(* IEC 61131-3 sources: SJ_AGV/PLC/Standard_functions.4.4.0/DataUpload, 2 files *)

(* ---- DataUpload_FB.ST ---- *)
FUNCTION_BLOCK DataUpload_FB
VAR_EXTERNAL
ndc8 : NDC8_T;

UploadData_ModBus_ValueWord:ARRAY[1..500] OF Word;
UploadData_ModBus_ValueBOOL:ARRAY[1..400] OF BOOL;

ConvWord:WORD;			(*Sum of the two first bytes*)

ConvByteL:Byte;			(*Low byte*)
ConvByteH:Byte;			(*High byte*)

ConvBit0:BOOL;			(*		 1 	    *)
ConvBit1:BOOL;			(*		 2 		*)
ConvBit2:BOOL;			(*		 4 		*)
ConvBit3:BOOL;			(*		 8 		*)
ConvBit4:BOOL;			(*	    10 		*)
ConvBit5:BOOL;			(*	    20 		*)
ConvBit6:BOOL;			(*	    40 		*)
ConvBit7:BOOL;          (*	    80 		*)
ConvBit8:BOOL;			(*		100     *)
ConvBit9:BOOL;			(*		200 	*)
ConvBit10:BOOL;			(*		400  	*)
ConvBit11:BOOL;			(*		800 	*)
ConvBit12:BOOL;			(*	   1000 	*)
ConvBit13:BOOL;			(*	   2000 	*)
ConvBit14:BOOL;			(*	   4000 	*)
ConvBit15:BOOL;         (*	   8000 	*)

(*BeijerSetParameters:BeijerSetParameters_T;*)

END_VAR

VAR_INPUT

END_VAR

VAR_OUTPUT

END_VAR

VAR

Angle_DINT : DINT;
Angle_REAL : REAL;

DataUpload : DataUpload_ModbusTCPIP_FB;

END_VAR
(****************************************************************************)

(* Update Data *)

(* Scanner_x *)
ConvDINT := NDC8.LS2000.X;
UploadData_ModBus_ValueWord [2]:=ConvWord2;
UploadData_ModBus_ValueWord [1]:=ConvWord;

(* Scanner_y *)
ConvDINT := NDC8.LS2000.Y;
UploadData_ModBus_ValueWord [4]:=ConvWord2;
UploadData_ModBus_ValueWord [3]:=ConvWord;

(* Scanner_t *)
Angle_REAL := NDC8.LS2000.Angle * 100.0;
Angle_DINT := REAL_TO_DINT(Angle_REAL);

ConvDINT := Angle_DINT;
UploadData_ModBus_ValueWord [6]:=ConvWord2;
UploadData_ModBus_ValueWord [5]:=ConvWord;

(* Max Speed *)
ConvDINT := NDC8.Vehicle.MaxSpeed;
UploadData_ModBus_ValueWord [8]:=ConvWord2;
UploadData_ModBus_ValueWord [7]:=ConvWord;

(* Enc1Scal *)
ConvUDINT := NDC8.DCD_6.SteerEncScale;
UploadData_ModBus_ValueWord [10]:=ConvWord2;
UploadData_ModBus_ValueWord [9]:=ConvWord;

(* Enc1Offs *)
ConvDINT := INT_TO_DINT(NDC8.DCD_6.SteerEncOffset);
UploadData_ModBus_ValueWord [12]:=ConvWord2;
UploadData_ModBus_ValueWord [11]:=ConvWord;

(* Enc3Scal *)
ConvUDINT := NDC8.DCD_8.SteerEncScale;
UploadData_ModBus_ValueWord [14]:=ConvWord2;
UploadData_ModBus_ValueWord [13]:=ConvWord;

(* Enc3Offs *)
ConvDINT := INT_TO_DINT(NDC8.DCD_8.SteerEncOffset);
UploadData_ModBus_ValueWord [16]:=ConvWord2;
UploadData_ModBus_ValueWord [15]:=ConvWord;

(* Enc2Scal *)
ConvUDINT := NDC8.DCD_5.DriveEncScale;
UploadData_ModBus_ValueWord [18]:=ConvWord2;
UploadData_ModBus_ValueWord [17]:=ConvWord;

(* Enc4Scal *)
ConvUDINT := NDC8.DCD_7.DriveEncScale;
UploadData_ModBus_ValueWord [20]:=ConvWord2;
UploadData_ModBus_ValueWord [19]:=ConvWord;

(* Batt Low Voltage *)
ConvDINT := NDC8.UserDefined.Integer32_50_BattLowVol;
UploadData_ModBus_ValueWord [22]:=ConvWord2;
UploadData_ModBus_ValueWord [21]:=ConvWord;

(* TravelDistance *)
ConvDINT := NDC8.UserDefined.Integer32_55_TravelDistance;
UploadData_ModBus_ValueWord [28]:=ConvWord2;
UploadData_ModBus_ValueWord [27]:=ConvWord;

(* LS2000 used Time Min *)
ConvDINT := NDC8.UserDefined.Integer32_60_LS2000_Attached_M;
UploadData_ModBus_ValueWord [30]:=ConvWord2;
UploadData_ModBus_ValueWord [29]:=ConvWord;

(* LS2000 used Time Hour *)
ConvDINT := NDC8.UserDefined.Integer32_59_LS2000_Attached_H;
UploadData_ModBus_ValueWord [32]:=ConvWord2;
UploadData_ModBus_ValueWord [31]:=ConvWord;

(* LS2000 used Time Day *)
ConvDINT := NDC8.UserDefined.Integer32_58_LS2000_Attached_D;
UploadData_ModBus_ValueWord [34]:=ConvWord2;
UploadData_ModBus_ValueWord [33]:=ConvWord;

(* Navigation Level *)
ConvDINT := NDC8.Position.NavLevel;
UploadData_ModBus_ValueWord [36]:=ConvWord2;
UploadData_ModBus_ValueWord [35]:=ConvWord;

(* AGV Drive Mode *)
UploadData_ModBus_ValueWord [41] := DINT_TO_WORD(Input.SteerMode);

(* Front Drive Current *)
UploadData_ModBus_ValueWord [42] := INT_TO_WORD(NDC8.DCD_5.TorqueCurrentReference);

(* Front Steer Current *)
UploadData_ModBus_ValueWord [43] := INT_TO_WORD(NDC8.DCD_6.TorqueCurrentReference);

(* Rear Drive Current *)
UploadData_ModBus_ValueWord [44] := INT_TO_WORD(NDC8.DCD_7.TorqueCurrentReference);

(* Rear Steer Current *)
UploadData_ModBus_ValueWord [45] := INT_TO_WORD(NDC8.DCD_8.TorqueCurrentReference);

(* Drive Current Diff*)
(*
UploadData_ModBus_ValueWord [46] := INT_TO_WORD(NDC8.DCD_5.TorqueCurrentReference - NDC8.DCD_7.TorqueCurrentReference);
*)
(* Steer Current Diff*)
(*
UploadData_ModBus_ValueWord [47] := INT_TO_WORD(NDC8.DCD_6.TorqueCurrentReference - NDC8.DCD_8.TorqueCurrentReference);
*)

(* Set Parameters *)
if UploadData_ModBus_ValueWord [71] <> 0 then
	(* Scanner_x *)
	ConvWord2 := UploadData_ModBus_ValueWord [73];
	ConvWord := UploadData_ModBus_ValueWord [72];

	NDC8.LS2000.X := ConvDINT;

	(* Scanner_y *)
	ConvWord2 := UploadData_ModBus_ValueWord [75];
	ConvWord := UploadData_ModBus_ValueWord [74];

	NDC8.LS2000.Y := ConvDINT;

	(* Scanner_t *)
	ConvWord2 := UploadData_ModBus_ValueWord [77];
	ConvWord := UploadData_ModBus_ValueWord [76];

	Angle_DINT := ConvDINT;

	Angle_REAL := DINT_TO_REAL(Angle_DINT) / 100.0;

	NDC8.LS2000.Angle := Angle_REAL;

	(* Max Speed *)
	ConvWord2 := UploadData_ModBus_ValueWord [79];
	ConvWord := UploadData_ModBus_ValueWord [78];

	NDC8.Vehicle.MaxSpeed := ConvDINT;

	(* Enc1Scal *)
	ConvWord2 := UploadData_ModBus_ValueWord [81];
	ConvWord := UploadData_ModBus_ValueWord [80];

	NDC8.DCD_6.SteerEncScale := ConvUDINT;

	(* Enc1Offs *)
	ConvWord2 := UploadData_ModBus_ValueWord [83];
	ConvWord := UploadData_ModBus_ValueWord [82];

	NDC8.DCD_6.SteerEncOffset := DINT_TO_INT(ConvDINT);

	(* Enc3Scal *)
	ConvWord2 := UploadData_ModBus_ValueWord [85];
	ConvWord := UploadData_ModBus_ValueWord [84];

	NDC8.DCD_8.SteerEncScale := ConvUDINT;

	(* Enc3Offs *)
	ConvWord2 := UploadData_ModBus_ValueWord [87];
	ConvWord := UploadData_ModBus_ValueWord [86];

	NDC8.DCD_8.SteerEncOffset := DINT_TO_INT(ConvDINT);

	(* Enc2Scal *)
	ConvWord2 := UploadData_ModBus_ValueWord [89];
	ConvWord := UploadData_ModBus_ValueWord [88];

	NDC8.DCD_5.DriveEncScale := ConvUDINT;

	(* Enc4Scal *)
	ConvWord2 := UploadData_ModBus_ValueWord [91];
	ConvWord := UploadData_ModBus_ValueWord [90];

	NDC8.DCD_7.DriveEncScale := ConvUDINT;

	(* Batt Low Voltage *)
	ConvWord2 := UploadData_ModBus_ValueWord [93];
	ConvWord := UploadData_ModBus_ValueWord [92];

	NDC8.UserDefined.Integer32_50_BattLowVol := ConvDINT;

	(*UploadData_ModBus_ValueBOOL [1] := FALSE;*)
end_if;

(****************************************************************************)
(*		Required for sending data to the display							*)

DataUpload();

(****************************************************************************)

END_FUNCTION_BLOCK

(* ---- DataUpload_ModbusTCPIP_FB.ST ---- *)
FUNCTION_BLOCK DATAUPLOAD_MODBUSTCPIP_FB
VAR_EXTERNAL
ndc8 : NDC8_T;

UploadData_ModBus_ValueWord:ARRAY[1..500] OF Word;
UploadData_ModBus_ValueBOOL:ARRAY[1..400] OF BOOL;

ConvWord:WORD;			(*Sum of the two first bytes*)

ConvByteL:Byte;			(*Low byte*)
ConvByteH:Byte;			(*High byte*)

ConvBit0:BOOL;			(*		 1 	    *)
ConvBit1:BOOL;			(*		 2 		*)
ConvBit2:BOOL;			(*		 4 		*)
ConvBit3:BOOL;			(*		 8 		*)
ConvBit4:BOOL;			(*	    10 		*)
ConvBit5:BOOL;			(*	    20 		*)
ConvBit6:BOOL;			(*	    40 		*)
ConvBit7:BOOL;          (*	    80 		*)
ConvBit8:BOOL;			(*		100     *)
ConvBit9:BOOL;			(*		200 	*)
ConvBit10:BOOL;			(*		400  	*)
ConvBit11:BOOL;			(*		800 	*)
ConvBit12:BOOL;			(*	   1000 	*)
ConvBit13:BOOL;			(*	   2000 	*)
ConvBit14:BOOL;			(*	   4000 	*)
ConvBit15:BOOL;         (*	   8000 	*)

(*BeijerSetParameters:BeijerSetParameters_T;*)
END_VAR

VAR_INPUT

END_VAR

VAR_OUTPUT

END_VAR

VAR
serial_read : NDC8_SERIAL_READ;
serial_write : NDC8_SERIAL_WRITE;
init : BOOL := TRUE;
TOTAL : DINT;
tx_header_length : BYTE := 6;
dummy : BOOL;
tr_cmd : DINT;

start_adress : INT;

ProcStep,
ReadCounter,
DebugCounter		: DINT;
StartDelayTOF	: TOF;
StartDelay 		: BOOL;

X: INT;
Y: INT;
Z: INT;
End:INT;
Index:DINT;
debug1 :INT;
debug2 :INT;
tr_len : DINT;
num_words : DINT;
num_Byte : DINT;
num_Bit : DINT;
Extra:DINT;
length : DINT;
tx_length : BYTE;
ENDBIT:DINT;
debugByte :Byte;

dataindex : INT;
msg_index: INT;
ix : INT;
UploadData_message : ARRAY[1..300] of BYTE;

END_VAR
(****************************************************************************)
(*StartDelayTOF(IN:=StartDelay, PT:=t#20ms);*)

if init then
	serial_read.port := 'COM6';
	serial_write.port := 'COM6';
	init := false;
end_if;

(****************************************************************************)

		(* Only read every 20ms *)
case ProcStep of
0:
	    StartDelay:=False;
		(*IF Not StartDelayTOF.Q THEN*)
		    ProcStep:=1;
		(*END_IF; *)

(****************************************************************************)
1:

	serial_read();
	msg_index := 0;
	while serial_read.length > 0 do

		(* Copy message to local buffer *)
		for dataindex := 1 to serial_read.length by 1 do
			ix := dataindex + msg_index;
			UploadData_message[ix] := serial_read.data[dataindex];
		end_for;
		(* Point for next possible message *)
		msg_index := msg_index + serial_read.length;
		serial_read();
	end_while;

	IF msg_index <> 0 then
		ProcStep:=2;
	Else
		ProcStep:=0;
	END_IF;

(****************************************************************************)
2:
		    (* Parse *)
			tr_cmd := BYTE_TO_DINT(UploadData_message[8]);
			tr_len := BYTE_TO_DINT(UploadData_message[6]);

			dummy := TRACE_DINT('Cmd', tr_cmd);
			dummy := TRACE_DINT('Len', tr_len);

			(* Copy header *)
			serial_write.data[1] := UploadData_message[1];
			serial_write.data[2] := UploadData_message[2];
			serial_write.data[3] := UploadData_message[3];
			serial_write.data[4] := UploadData_message[4];
			serial_write.data[5] := UploadData_message[5];

			serial_write.data[6] := UploadData_message[6]; 	(* Length, will be overwritten *)
			serial_write.data[7] := UploadData_message[7]; 	(* Slave adress *)
			serial_write.data[8] := UploadData_message[8]; 	(* Cmd *)
			(* Start adress to read *)
			ConvByteH:= UploadData_message[9];
			ConvByteL:= UploadData_message[10];
			start_adress  := Word_TO_INT(ConvWord) + 1;
			ProcStep:=3;

(****************************************************************************)
3:

			(*Check Function type *)

			case tr_cmd of
				1: 	ProcStep:=10;	(* Check if Read Coils *)
				5:	ProcStep:=50;	(* Check if Write single Coil *)
				15:	ProcStep:=150;	(* Check if Write Multiple Coils *)
				6:	ProcStep:=60;	(* Check if Write single register *)
				16:	ProcStep:=160; (* Check if write Multiple register *)
				3:	ProcStep:=30;	(*Check if Read register *)
			Else
				ProcStep:=999; 	(*Send Echo *)
			end_case;

(****************************************************************************)
10:
					(* Read Coils *)
					(* Number of Bits *)
				(* serial_read.data[11]; *)
				ConvByteH:= UploadData_message[11];
				ConvByteL:= UploadData_message[12];
				num_Bit  := Word_TO_DINT(ConvWord);
				num_Byte :=(num_Bit/8)+1;
				ENDBIT:=(num_Bit/8);
				Extra:=num_Bit-ENDBIT;
					Y:=start_adress;
					Z:=10;
					Serial_write.data[9] := DINT_TO_BYTE(num_Byte);

				 IF  ENDBIT<>0 THEN
					For Index:=1 to ENDBIT BY 1 DO

						ConvBit0:=UploadData_ModBus_ValueBOOL [Y];
						Y:=Y+1;
						ConvBit1:=UploadData_ModBus_ValueBOOL [Y];
						Y:=Y+1;
						ConvBit2:=UploadData_ModBus_ValueBOOL [Y];
						Y:=Y+1;
						ConvBit3:=UploadData_ModBus_ValueBOOL [Y];
						Y:=Y+1;
						ConvBit4:=UploadData_ModBus_ValueBOOL [Y];
						Y:=Y+1;
						ConvBit5:=UploadData_ModBus_ValueBOOL [Y];
						Y:=Y+1;
						ConvBit6:=UploadData_ModBus_ValueBOOL [Y];
						Y:=Y+1;
						ConvBit7:=UploadData_ModBus_ValueBOOL [Y];
						serial_write.data[Z]:=ConvByteL;
						Y:=Y+1;
						Z:=Z+1;
					END_FOR;
				END_IF;

				(*Fill in last Byte *)
				IF Extra <> 0 Then
					ConvByteL:=0;

					   	  ConvBit0:=UploadData_ModBus_ValueBOOL [Y];
					If Extra >1 Then
						Y:=Y+1;
						ConvBit1:=UploadData_ModBus_ValueBOOL [Y];
					END_IF;
					If Extra >2 Then
						Y:=Y+1;
						ConvBit2:=UploadData_ModBus_ValueBOOL [Y];
					END_IF;
					If Extra >3 Then
						Y:=Y+1;
						ConvBit3:=UploadData_ModBus_ValueBOOL [Y];
					END_IF;
					If Extra >4 Then
						Y:=Y+1;
						ConvBit4:=UploadData_ModBus_ValueBOOL [Y];
					END_IF;
					If Extra >5 Then
						Y:=Y+1;
						ConvBit5:=UploadData_ModBus_ValueBOOL [Y];
					END_IF;
					If Extra >6 Then
						Y:=Y+1;
						ConvBit6:=UploadData_ModBus_ValueBOOL [Y];
					END_IF;
					serial_write.data[Z]:=ConvByteL;

				END_IF;

					length := num_Byte+3;
					tx_length := DINT_TO_BYTE(length);
					serial_write.data[6] := tx_length; (* lp *)
					ProcStep:=10000;

(****************************************************************************)
30:
						(*Read register *)
						(* Number of words *)
					UploadData_ModBus_ValueWord [46] := PLC_TX_Word1;
					UploadData_ModBus_ValueWord [47] := PLC_TX_Word2;
					UploadData_ModBus_ValueWord [48] := PLC_TX_Word3;
					UploadData_ModBus_ValueWord [49] := PLC_TX_Word4;
					UploadData_ModBus_ValueWord [50] := PLC_TX_Word5;
					UploadData_ModBus_ValueWord [51] := PLC_TX_Word6;
					UploadData_ModBus_ValueWord [52] := PLC_TX_Word7_STr_Vecl;
					UploadData_ModBus_ValueWord [53] := PLC_TX_Word8_STr_Seg;
					UploadData_ModBus_ValueWord [54] := PLC_TX_Word9_STr_Pnt;
					UploadData_ModBus_ValueWord [55] := PLC_TX_Word10_STr_BatV;
					UploadData_ModBus_ValueWord [56] := PLC_TX_Word11_STr_Temp;
					UploadData_ModBus_ValueWord [57] := PLC_TX_Word12_STr_BatD;
					UploadData_ModBus_ValueWord [58] := PLC_TX_Word13_STr_Err;
					UploadData_ModBus_ValueWord [59] := PLC_TX_Word14_STr_BCD3;
					UploadData_ModBus_ValueWord [60] := PLC_TX_Word15_STr_BCD2;
					UploadData_ModBus_ValueWord [61] := PLC_TX_Word16_STr_BCD1;
					num_words := BYTE_TO_DINT(UploadData_message[12]);
					Total := num_words;
					Y := start_adress;
					(* Copy header *)
					serial_write.data[1] := UploadData_message[1];
					serial_write.data[2] := UploadData_message[2];
					serial_write.data[3] := UploadData_message[3];
					serial_write.data[4] := UploadData_message[4];
					serial_write.data[5] := UploadData_message[5];
					Z:= 1; (* Send first 9*)
					serial_write.data[6] := DINT_TO_BYTE(Total*2 + 3); (* lp *)
					serial_write.data[7] := UploadData_message[7]; 	(* Slave adress *)
					serial_write.data[8] := UploadData_message[8]; 	(* Cmd *)
					serial_write.data[9] := DINT_TO_BYTE(Total*2); (* lp *)
				    serial_write.length := 9;
					serial_write();
					if PLC_TX04_Bit_ChkCom_Tx = true then
						PLC_TX04_Bit_ChkCom_Tx := false;
					else
						PLC_TX04_Bit_ChkCom_Tx := true;
					end_if;
					ProcStep:=31;
31:
					IF Total >= 16 THEN
						Total := Total - 16;
					For Index:=1 to 16 BY 1 DO
						ConvWord:=UploadData_ModBus_ValueWord [Y];
						serial_write.data[Z]:=ConvByteH;
						Z:=Z+1;
						serial_write.data[Z]:=ConvByteL;
						Z:=Z+1;
						Y:=Y+1;
					END_FOR;
					serial_write.length := DINT_TO_INT(32); (*Will be max 32 bytes*)
					serial_write();
					Z := 1;
					ProcStep:=31;
					ELSIF Total = 0 THEN
						ProcStep:=10001;
					ELSE
					For Index:=1 to (TOTAL) BY 1 DO
						ConvWord:=UploadData_ModBus_ValueWord [Y];
						serial_write.data[Z]:=ConvByteH;
						Z:=Z+1;
						serial_write.data[Z]:=ConvByteL;
						Z:=Z+1;
						Y:=Y+1;
					END_FOR;
					serial_write.length := DINT_TO_INT(TOTAL*2);
					serial_write();
					Z := 1;
					ProcStep:=10001;
					END_IF;
(****************************************************************************)
50:
			(* Write single Coil *)

					Y:=start_adress;
					ConvByteL := UploadData_message[11];
					UploadData_ModBus_ValueBOOL [Y]:= ConvBit0;

					ProcStep:=999;

	(****************************************************************************)
60:
				(* Write single register *)
				(* single write *)
				(* Number of words *)
				(* serial_read.data[11]; *)
				num_words := BYTE_TO_DINT(UploadData_message[12]);
				Y:=start_adress;
				ConvByteH:=UploadData_message[11];
			    ConvByteL:=UploadData_message[12];
				UploadData_ModBus_ValueWord [Y]:=ConvWord;

				ProcStep:=999;

(****************************************************************************)
150:
					(*Write Multiple Coils  *)
					(* Number of Bits *)
				(* serial_read.data[11]; *)
				ConvByteH:= UploadData_message[11];
				ConvByteL:= UploadData_message[12];
				num_Bit  := Word_TO_DINT(ConvWord);
				num_Byte :=(num_Bit/8)+1;
				ENDBIT:=(num_Bit/8);
				Extra:=num_Bit-ENDBIT;
					Y:=start_adress;
					Z:=10;

				 IF  ENDBIT <>0 THEN
					For Index:=1 to ENDBIT BY 1 DO

						ConvByteL:= UploadData_message[Z];
						UploadData_ModBus_ValueBOOL [Y]:=ConvBit0;
						Y:=Y+1;
						UploadData_ModBus_ValueBOOL [Y]:=ConvBit1;
						Y:=Y+1;
						UploadData_ModBus_ValueBOOL [Y]:=ConvBit2;
						Y:=Y+1;
						UploadData_ModBus_ValueBOOL [Y]:=ConvBit3;
						Y:=Y+1;
						UploadData_ModBus_ValueBOOL [Y]:=ConvBit4;
						Y:=Y+1;
						UploadData_ModBus_ValueBOOL [Y]:=ConvBit5;
						Y:=Y+1;
						UploadData_ModBus_ValueBOOL [Y]:=ConvBit6;
						Y:=Y+1;
						UploadData_ModBus_ValueBOOL [Y]:=ConvBit7;
						Y:=Y+1;
						Z:=Z+1;
					END_FOR;
				END_IF;

				(*Fill in last Bits *)
				ConvByteL:= UploadData_message[Z];
				IF Extra <> 0 Then
					UploadData_ModBus_ValueBOOL [Y]:=ConvBit0;
					If Extra >1 Then
						Y:=Y+1;
						UploadData_ModBus_ValueBOOL [Y]:=ConvBit1;
					END_IF;
					If Extra >2 Then
						Y:=Y+1;
						UploadData_ModBus_ValueBOOL [Y]:=ConvBit2;
					END_IF;
					If Extra >3 Then
						Y:=Y+1;
						UploadData_ModBus_ValueBOOL [Y]:=ConvBit3;
					END_IF;
					If Extra >4 Then
						Y:=Y+1;
						UploadData_ModBus_ValueBOOL [Y]:=ConvBit4;
					END_IF;
					If Extra >5 Then
						Y:=Y+1;
						UploadData_ModBus_ValueBOOL [Y]:=ConvBit5;
					END_IF;
					If Extra >6 Then
						Y:=Y+1;
						UploadData_ModBus_ValueBOOL [Y]:=ConvBit6;
					END_IF;

				END_IF;
				ProcStep:=999;

(****************************************************************************)
160:
				(* Multiple write *)
				num_words:=Byte_TO_DInt(UploadData_message[12]);
				(* Check if message lenght outside the Buffer, if so do what ??? *)
			(*	IF num_words > 9 THEN
				   num_words:=9;
				END_IF;    *)
				Y:=start_adress;
				X:=14;
				End:= Byte_TO_Int(UploadData_message[12]);

				For Index:=1 to num_words BY 1 DO
					ConvByteH:=UploadData_message[X];
					X:=X+1;
					ConvByteL:=UploadData_message[X];
					UploadData_ModBus_ValueWord [Y]:=ConvWord;
					X:=X+1;
					Y:=Y+1;
				END_FOR;
						(*Set Into Memory *)
		PLC_RX_Word1 := UploadData_ModBus_ValueWord [94];
		PLC_RX_Word2 := UploadData_ModBus_ValueWord [95];
		PLC_RX_Word3 := UploadData_ModBus_ValueWord [96];
		PLC_RX_Word4 := UploadData_ModBus_ValueWord [97];
		PLC_RX_Word5 := UploadData_ModBus_ValueWord [98];
		PLC_RX_Word6 := UploadData_ModBus_ValueWord [99];
		PLC_RX_Word7_STw_BCD3 := UploadData_ModBus_ValueWord [100];
		PLC_RX_Word8_STw_BCD2 := UploadData_ModBus_ValueWord [101];
		PLC_RX_Word9_STw_BCD1 := UploadData_ModBus_ValueWord [102];
		PLC_RX_Word10_STw_ILEr := UploadData_ModBus_ValueWord [103];
		PLC_RX_Word11_Ins_Pno := UploadData_ModBus_ValueWord [104];
		PLC_RX_Word12_STw_Pint := UploadData_ModBus_ValueWord [105];
		PLC_RX_Word13_Ins_Ano := UploadData_ModBus_ValueWord [106];
		PLC_RX_Word14_BMS_2 := UploadData_ModBus_ValueWord [107];
		PLC_RX_Word15_BMS_3 := UploadData_ModBus_ValueWord [108];
		PLC_RX_Word16_BMS_BatV := UploadData_ModBus_ValueWord [109];
		PLC_RX_Word17_BMS_BatT := UploadData_ModBus_ValueWord [110];
		PLC_RX_Word18_BMS_BatC := UploadData_ModBus_ValueWord [111];
		PLC_RX_Word19_BMS_BatA := UploadData_ModBus_ValueWord [112];
		PLC_RX_Word20_PLC_ErrD := UploadData_ModBus_ValueWord [113];
		PLC_RX_Word21_BMS_Main := UploadData_ModBus_ValueWord [114];
		PLC_RX_Word22_BMS_Chan := UploadData_ModBus_ValueWord [115];
		PLC_RX_Word23_BMS_ID4L := UploadData_ModBus_ValueWord [116];
		PLC_RX_Word24_BMS_ID4H := UploadData_ModBus_ValueWord [117];
	PLC_RX_Word25 := UploadData_ModBus_ValueWord [118];
				ProcStep:=998;
998:
				Serial_write.data[1] := UploadData_message[1];
				Serial_write.data[2] := UploadData_message[2];
				Serial_write.data[3] := UploadData_message[3];
				Serial_write.data[4] := UploadData_message[4];
				Serial_write.data[5] := UploadData_message[5];
				Serial_write.data[6] := DINT_TO_BYTE(6);
				Serial_write.data[7] := UploadData_message[7];
				Serial_write.data[8] := UploadData_message[8];
				Serial_write.data[9] := UploadData_message[9];
				serial_write.data[10] := UploadData_message[10];
				serial_write.data[11] := UploadData_message[11];
				serial_write.data[12] := UploadData_message[12];  (*PLC_message[12];*)
				serial_write.length := 12;
				serial_write();
				ProcStep:=10001;
(****************************************************************************)
999:

				(*Send Echo *)
					Serial_write.data[9] := UploadData_message[9];
					serial_write.data[10] := UploadData_message[10];
					serial_write.data[11] := UploadData_message[11];
					serial_write.data[12] := UploadData_message[12];

					length :=6;
					tx_length := DINT_TO_BYTE(length);
			        serial_write.data[6] := tx_length; (* lp *)
					ProcStep:=10000;

(****************************************************************************)
10000:

			(*Send Data *)

			serial_write.length := BYTE_TO_INT(tx_header_length) + BYTE_TO_INT(tx_length);
			serial_write();

			serial_write.length := 0;
			serial_write();

			IF serial_write.sent<>0 or serial_write.error<>0 Then
				ProcStep:=0;
				DebugCounter := DebugCounter + 1;
			End_IF;
(****************************************************************************)
10001:
			serial_write.length := 0; (*Using SendBuffer =1 length needs to be set to 0 for it to be sent*)
			serial_write(); (*send*)
			IF serial_write.sent<>0 or serial_write.error<>0 Then
				ProcStep:=0;
				DebugCounter := DebugCounter + 1;
			End_IF;
			ProcStep:=0;
end_case;

END_FUNCTION_BLOCK
